(* Schneider Machine Expert - Basic project Imam Pratama Setiady, file version 1.7.0.0 *)
(* ProjectInformations: Name=New project *)

HARDWARE
  Cpu 0: TM221ME32TK
  EthernetConfiguration: NetworkName=M221, IpAllocationMode=FixedAddress, IpAddress=0.0.0.0, SubnetMask=0.0.0.0
  SerialLineConfiguration: Baud=Baud19200, Parity=ParityEven, DataBits=DataBits8, StopBits=StopBits1, PhysicalMedium=PhysicalMediumRs485, TransmissionMode=TransmissionModeModbusRtu, SlaveId=1, Addressing=SlaveAddressing
  MastTask: UsePeriodScanMode=false, PeriodScan=100
  FastTask: Period=255
  CpuBehavior: StartingMode=StartAsPreviousState, AutoSaveRamOnEeprom=true, WatchdogPeriod=250

SYMBOLS  (address, symbol, comment, settings)
  %TM1        [Preset=5, Base=OneSecond]
  %TM2        [Preset=5, Base=OneSecond]
  %TM3        [Preset=5, Base=OneSecond]
  %TM4        [Preset=5, Base=OneSecond]
  %TM5        [Preset=5, Base=OneSecond]
  %TM6        [Preset=5, Base=OneSecond]
  %TM7        [Preset=5, Base=OneSecond]
  %TM8        [Preset=5, Base=OneSecond]
  %Q0.0       "Merah 1"
  %Q0.1       "Kuning 1"
  %Q0.2       "Hijau 1"
  %Q0.3       "Merah 2"
  %Q0.4       "Kuning 2"
  %Q0.5       "Hijau 2"
  %Q0.6       "Merah 3"
  %Q0.7       "Kuning 3"
  %Q0.8       "Hijau 3"
  %Q0.9       "Merah 4"
  %Q0.10      "Kuning 4"
  %Q0.11      "Hijau 4"

POU New POU
  (* SectionNumber=1 *)

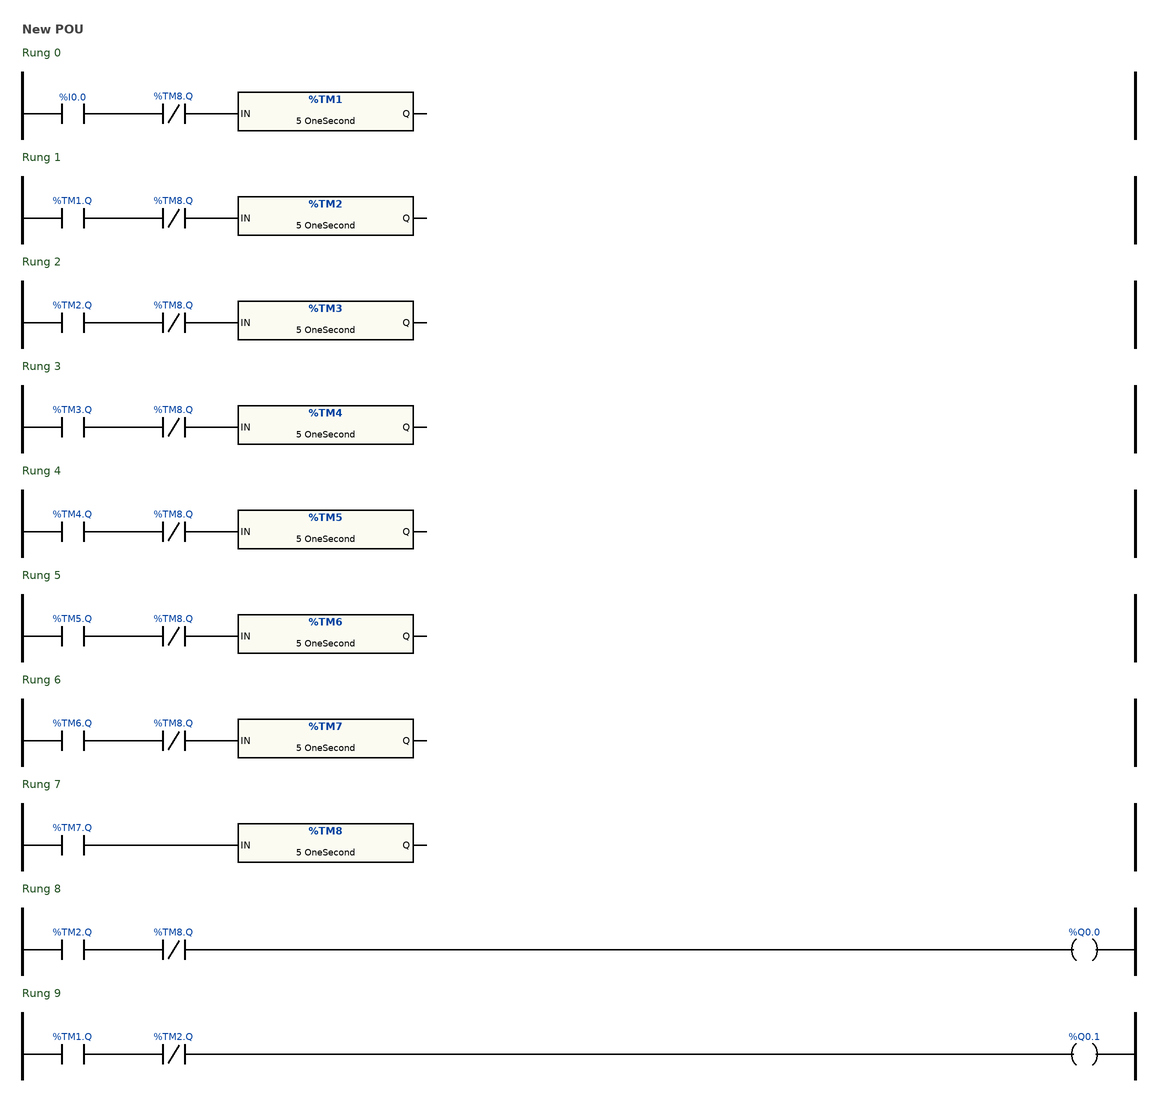

// Rung 0
  BLK %TM1
  LD %I0.0
  ANDN %TM8.Q
  IN
  END_BLK
  // as ST:
  //   %TM1(IN := %I0.0 AND NOT %TM8.Q);

// Rung 1
  BLK %TM2
  LD %TM1.Q
  ANDN %TM8.Q
  IN
  END_BLK
  // as ST:
  //   %TM2(IN := %TM1.Q AND NOT %TM8.Q);

// Rung 2
  BLK %TM3
  LD %TM2.Q
  ANDN %TM8.Q
  IN
  END_BLK
  // as ST:
  //   %TM3(IN := %TM2.Q AND NOT %TM8.Q);

// Rung 3
  BLK %TM4
  LD %TM3.Q
  ANDN %TM8.Q
  IN
  END_BLK
  // as ST:
  //   %TM4(IN := %TM3.Q AND NOT %TM8.Q);

// Rung 4
  BLK %TM5
  LD %TM4.Q
  ANDN %TM8.Q
  IN
  END_BLK
  // as ST:
  //   %TM5(IN := %TM4.Q AND NOT %TM8.Q);

// Rung 5
  BLK %TM6
  LD %TM5.Q
  ANDN %TM8.Q
  IN
  END_BLK
  // as ST:
  //   %TM6(IN := %TM5.Q AND NOT %TM8.Q);

// Rung 6
  BLK %TM7
  LD %TM6.Q
  ANDN %TM8.Q
  IN
  END_BLK
  // as ST:
  //   %TM7(IN := %TM6.Q AND NOT %TM8.Q);

// Rung 7
  BLK %TM8
  LD %TM7.Q
  IN
  END_BLK
  // as ST:
  //   %TM8(IN := %TM7.Q);

// Rung 8
  LD %TM2.Q
  ANDN %TM8.Q
  ST %Q0.0
  // as ST:
  //   %Q0.0 := %TM2.Q AND NOT %TM8.Q;

// Rung 9
  LD %TM1.Q
  ANDN %TM2.Q
  ST %Q0.1
  // as ST:
  //   %Q0.1 := %TM1.Q AND NOT %TM2.Q;

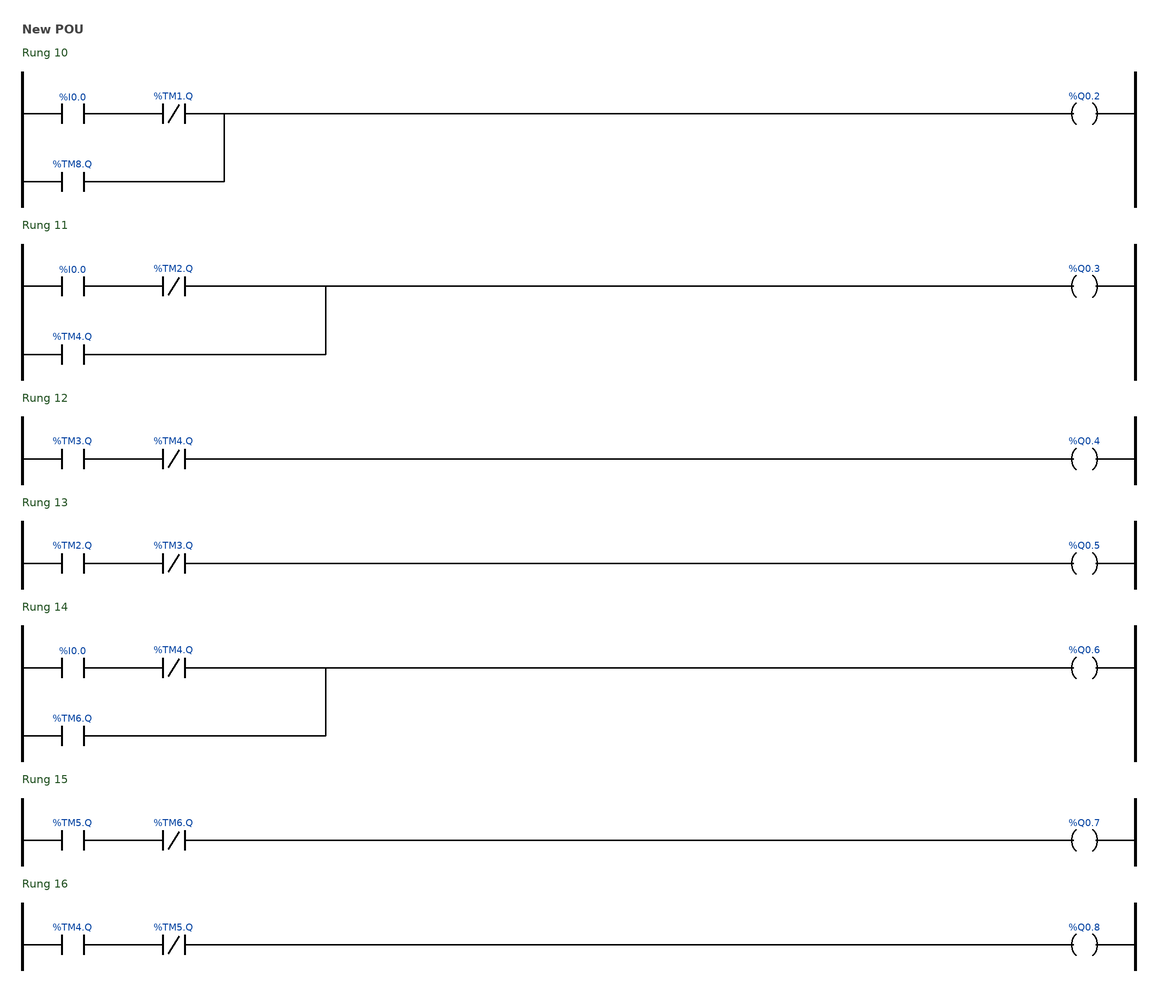

// Rung 10
  LD %I0.0
  ANDN %TM1.Q
  OR %TM8.Q
  ST %Q0.2
  // as ST:
  //   %Q0.2 := %I0.0 AND NOT %TM1.Q OR %TM8.Q;

// Rung 11
  LD %I0.0
  ANDN %TM2.Q
  OR %TM4.Q
  ST %Q0.3
  // as ST:
  //   %Q0.3 := %I0.0 AND NOT %TM2.Q OR %TM4.Q;

// Rung 12
  LD %TM3.Q
  ANDN %TM4.Q
  ST %Q0.4
  // as ST:
  //   %Q0.4 := %TM3.Q AND NOT %TM4.Q;

// Rung 13
  LD %TM2.Q
  ANDN %TM3.Q
  ST %Q0.5
  // as ST:
  //   %Q0.5 := %TM2.Q AND NOT %TM3.Q;

// Rung 14
  LD %I0.0
  ANDN %TM4.Q
  OR %TM6.Q
  ST %Q0.6
  // as ST:
  //   %Q0.6 := %I0.0 AND NOT %TM4.Q OR %TM6.Q;

// Rung 15
  LD %TM5.Q
  ANDN %TM6.Q
  ST %Q0.7
  // as ST:
  //   %Q0.7 := %TM5.Q AND NOT %TM6.Q;

// Rung 16
  LD %TM4.Q
  ANDN %TM5.Q
  ST %Q0.8
  // as ST:
  //   %Q0.8 := %TM4.Q AND NOT %TM5.Q;

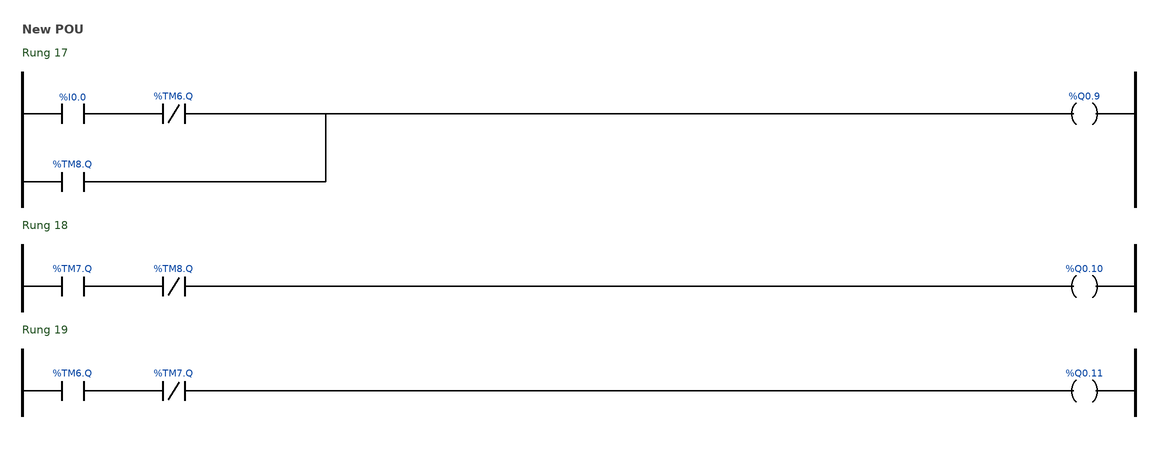

// Rung 17
  LD %I0.0
  ANDN %TM6.Q
  OR %TM8.Q
  ST %Q0.9
  // as ST:
  //   %Q0.9 := %I0.0 AND NOT %TM6.Q OR %TM8.Q;

// Rung 18
  LD %TM7.Q
  ANDN %TM8.Q
  ST %Q0.10
  // as ST:
  //   %Q0.10 := %TM7.Q AND NOT %TM8.Q;

// Rung 19
  LD %TM6.Q
  ANDN %TM7.Q
  ST %Q0.11
  // as ST:
  //   %Q0.11 := %TM6.Q AND NOT %TM7.Q;
